# EPICS autosave request: vici/viciUM_positions.req
$(P)$(Q):POSN.FRST
$(P)$(Q):POSN.FVST
$(P)$(Q):POSN.ONST
$(P)$(Q):POSN.SVST
$(P)$(Q):POSN.SXST
$(P)$(Q):POSN.THST
$(P)$(Q):POSN.TWST
$(P)$(Q):POSN.ZRST
$(P)$(Q):POSN:RBV.FRST
$(P)$(Q):POSN:RBV.FVST
$(P)$(Q):POSN:RBV.ONST
$(P)$(Q):POSN:RBV.SVST
$(P)$(Q):POSN:RBV.SXST
$(P)$(Q):POSN:RBV.THST
$(P)$(Q):POSN:RBV.TWST
$(P)$(Q):POSN:RBV.ZRST
